FUNCTION_BLOCK DOUBLE_SENSOR_ADCPI
  {SET_ATTRIBUTE(OpcUa, POINT.ENDPOINT)}
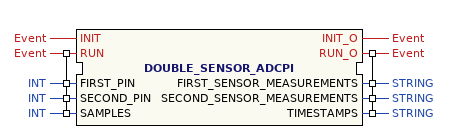
  EVENT_INPUT
    INIT;
    RUN WITH FIRST_PIN, SECOND_PIN, SAMPLES;
  END_EVENT
  EVENT_OUTPUT
    INIT_O;
    RUN_O WITH FIRST_SENSOR_MEASUREMENTS, SECOND_SENSOR_MEASUREMENTS, TIMESTAMPS;
  END_EVENT
  VAR_INPUT
    FIRST_PIN : INT; {SET_ATTRIBUTE(OpcUa, Variable)}
    SECOND_PIN : INT; {SET_ATTRIBUTE(OpcUa, Variable)}
    SAMPLES : INT; {SET_ATTRIBUTE(OpcUa, Variable)}
  END_VAR
  VAR_OUTPUT
    FIRST_SENSOR_MEASUREMENTS : STRING; {SET_ATTRIBUTE(OpcUa, Variable)}
    SECOND_SENSOR_MEASUREMENTS : STRING; {SET_ATTRIBUTE(OpcUa, Variable)}
    TIMESTAMPS : STRING; {SET_ATTRIBUTE(OpcUa, Variable)}
  END_VAR
END_FUNCTION_BLOCK
